{attribute 'GeneratedUsingTerminal: EL4031-0000-0016'}
{attribute addProperty BoxType "EL4031-0000-0016"}
{attribute addProperty Id "AO_OutputsAT %Q*AO_Outputs_BA7EBB7C2WcStateAT %I*WcState_0B2B16F91InfoDataAT %I*InfoData_94A18F5E2"}
{attribute addProperty CRC "3372769853"}
{attribute addProperty Size "5"}
TYPE EL4031_C908623D EXTENDS EtcSlaveTerminalBase_947E5A46 :
STRUCT
	{attribute addProperty Name "AO_Outputs"}
	AO_Outputs : AO_Outputs_BA7EBB7C;
	{attribute addProperty Name "WcState"}
	WcState : WcState_0B2B16F9;
	{attribute addProperty Name "InfoData"}
	InfoData : InfoData_94A18F5E;
END_STRUCT
END_TYPE

(* stored: Version 1.2.0.0, ProductVersion 3.1.4024.9
   DUT EL4031_C908623D: Id {ebfc656d-9c8b-4ce5-869d-94939185c526} *)
